// TIA Portal V20 export
ORGANIZATION_BLOCK "Startup"   // OB1040, LAD, Startup
TITLE = "Complete Restart"
AUTHOR : ERsystem_FA2_DH. Kim
// stored: AutoNumber false, IsIECCheckEnabled true, Namespace Unit1.Em4, SetENOAutomatically false
   VAR_INPUT
      LostRetentive : Bool;   // True if retentive data are lost
      LostRTC : Bool;   // True if date and time are lost
   END_VAR
BEGIN

REGION Network 1 (SCL): Build the Absolut Reference Designator
   // Set the Absoult Reference Designator in the Config DB
   IF LEN(IN := "Unit1.Em4.Config".em.referenceDesignator.parent) <> 0 THEN
     "Unit1.Em4.Config".em.referenceDesignator.combined := CONCAT_WSTRING(IN1 := "Unit1.Em4.Config".em.referenceDesignator.parent, IN2 := WSTRING#'.', IN3 := "Unit1.Em4.Config".em.referenceDesignator.relative);
   ELSE
     "Unit1.Em4.Config".em.referenceDesignator.combined := "Unit1.Em4.Config".em.referenceDesignator.relative;
   END_IF;
END_REGION

REGION Network 2 (SCL): Assign axes data
   //Assign axes
   "Unit1.Em4.Config".axis[1] := "BA040AZSCDR5_AnodeMainPnp1AxisX";
   "Unit1.Em4.Config".axis[2] := "BA040AZSCDR6_AnodeMainPnp2AxisX";
   "Unit1.Em4.Config".axis[3] := "BA040AZSCDR11_AnodeMainPnp1AxisY";
   "Unit1.Em4.Config".axis[4] := "BA040AZSCDR12_AnodeMainPnp1AxisZ";
   "Unit1.Em4.Config".axis[5] := "BA040AZSCDR14_AnodeMainPnp2AxisZ";
   "Unit1.Em4.Config".axis[6] := "BA040AZSCDR15_AnodeAlignTableAxisX";
   "Unit1.Em4.Config".axis[7] := "BA040AZSCDR16_AnodeAlignTableAxisY1";
   "Unit1.Em4.Config".axis[8] := "BA040AZSCDR17_AnodeAlignTableAxisY2";

   // Config.cam[1] := _.BA030AZSCDR5_AnodeMainPnp1AxisXCamMain;
   // Config.cam[2] := _.BA030AZSCDR6_AnodeMainPnp2AxisXCamMain;
   // Config.cam[3] := _.BA030AZSCDR12_AnodeMainPnp1AxisZCamMain;
   // Config.cam[4] := _.BA030AZSCDR14_AnodeMainPnp2AxisZCamMain;

   "Unit1.Em4.Config".outputCam[1] := "AnodePnP1XFwd";
   "Unit1.Em4.Config".outputCam[2] := "AnodePnP1XBwd";
   "Unit1.Em4.Config".outputCam[3] := "AnodePnP2XFwd";
   "Unit1.Em4.Config".outputCam[4] := "AnodePnP2XBwd";
   "Unit1.Em4.Config".outputCam[5] := "AnodePnPZ1Down1";
   "Unit1.Em4.Config".outputCam[6] := "AnodePnPZ1Up1";
   "Unit1.Em4.Config".outputCam[7] := "AnodePnPZ2Down1";
   "Unit1.Em4.Config".outputCam[8] := "AnodePnPZ2Up1";
   "Unit1.Em4.Config".outputCam[9] := "AnodePnPZ1Down2";
   "Unit1.Em4.Config".outputCam[10] := "AnodePnPZ1Up2";
   "Unit1.Em4.Config".outputCam[11] := "AnodePnPZ2Down2";
   "Unit1.Em4.Config".outputCam[12] := "AnodePnPZ2Up2";
   "Unit1.Em4.Config".outputCam[13] := "AnodePnPZ1SuctionOn";
   "Unit1.Em4.Config".outputCam[14] := "AnodePnPZ1SuctionOff";
   "Unit1.Em4.Config".outputCam[15] := "AnodePnPZ1ReelCutBlow";
   "Unit1.Em4.Config".outputCam[16] := "AnodePnPZ2SuctionOn";
   "Unit1.Em4.Config".outputCam[17] := "AnodePnPZ2SuctionOff";
   "Unit1.Em4.Config".outputCam[18] := "AnodeAlignSuctionOn";
   "Unit1.Em4.Config".outputCam[19] := "AnodeAlignSuctionOff";

   // Assign configuration data of axis

   // FB Enable
   "Unit1.Em4.HmiInterface".cmAnodeMainPnP1AxisX.commands.enableMasterControl := TRUE;
   "Unit1.Em4.HmiInterface".cmAnodeMainPnP1AxisY.commands.enableMasterControl := TRUE;
   "Unit1.Em4.HmiInterface".cmAnodeMainPnP1AxisZ.commands.enableMasterControl := TRUE;
   "Unit1.Em4.HmiInterface".cmAnodeMainPnP2AxisX.commands.enableMasterControl := TRUE;
   "Unit1.Em4.HmiInterface".cmAnodeMainPnP2AxisZ.commands.enableMasterControl := TRUE;
   "Unit1.Em4.HmiInterface".cmAnodeAlignTableAxisX.commands.enableMasterControl := TRUE;
   "Unit1.Em4.HmiInterface".cmAnodeAlignTableAxisY1.commands.enableMasterControl := TRUE;
   "Unit1.Em4.HmiInterface".cmAnodeAlignTableAxisY2.commands.enableMasterControl := TRUE;

   // Axis 1 BA030AZSCDR5_AnodeMainPnp1AxisX
   "Unit1.Em4.HmiInterface".cmAnodeMainPnP1AxisX.commandConfiguration.jog.velocity := 10.0;
   "Unit1.Em4.HmiInterface".cmAnodeMainPnP1AxisX.commandConfiguration.jog.acceleration := 100.0;
   "Unit1.Em4.HmiInterface".cmAnodeMainPnP1AxisX.commandConfiguration.jog.deceleration := 100.0;
   "Unit1.Em4.HmiInterface".cmAnodeMainPnP1AxisX.commandConfiguration.moveVelocity.velocity := 10.0;
   "Unit1.Em4.HmiInterface".cmAnodeMainPnP1AxisX.commandConfiguration.moveVelocity.acceleration := 100.0;
   "Unit1.Em4.HmiInterface".cmAnodeMainPnP1AxisX.commandConfiguration.moveVelocity.deceleration := 100.0;
   "Unit1.Em4.HmiInterface".cmAnodeMainPnP1AxisX.commandConfiguration.posRelative.velocity := 10.0;
   "Unit1.Em4.HmiInterface".cmAnodeMainPnP1AxisX.commandConfiguration.posRelative.acceleration := 100.0;
   "Unit1.Em4.HmiInterface".cmAnodeMainPnP1AxisX.commandConfiguration.posRelative.deceleration := 100.0;
   "Unit1.Em4.HmiInterface".cmAnodeMainPnP1AxisX.configuration.setPositions[0].name := 'reelCutConveyerPos';
   "Unit1.Em4.HmiInterface".cmAnodeMainPnP1AxisX.configuration.setPositions[1].name := 'alignTablePos';

   // Axis 2 BA030AZSCDR7_AnodeMainPnp2AxisX
   "Unit1.Em4.HmiInterface".cmAnodeMainPnP2AxisX.commandConfiguration.jog.velocity := 10.0;
   "Unit1.Em4.HmiInterface".cmAnodeMainPnP2AxisX.commandConfiguration.jog.acceleration := 100.0;
   "Unit1.Em4.HmiInterface".cmAnodeMainPnP2AxisX.commandConfiguration.jog.deceleration := 100.0;
   "Unit1.Em4.HmiInterface".cmAnodeMainPnP2AxisX.commandConfiguration.moveVelocity.velocity := 10.0;
   "Unit1.Em4.HmiInterface".cmAnodeMainPnP2AxisX.commandConfiguration.moveVelocity.acceleration := 100.0;
   "Unit1.Em4.HmiInterface".cmAnodeMainPnP2AxisX.commandConfiguration.moveVelocity.deceleration := 100.0;
   "Unit1.Em4.HmiInterface".cmAnodeMainPnP2AxisX.commandConfiguration.posRelative.velocity := 10.0;
   "Unit1.Em4.HmiInterface".cmAnodeMainPnP2AxisX.commandConfiguration.posRelative.acceleration := 100.0;
   "Unit1.Em4.HmiInterface".cmAnodeMainPnP2AxisX.commandConfiguration.posRelative.deceleration := 100.0;
   "Unit1.Em4.HmiInterface".cmAnodeMainPnP2AxisX.configuration.setPositions[0].name := 'alignTablePos';
   "Unit1.Em4.HmiInterface".cmAnodeMainPnP2AxisX.configuration.setPositions[1].name := 'stackTablePos';

   // Axis 3 BA030AZSCDR9_AnodeMainPnp1AxisY
   "Unit1.Em4.HmiInterface".cmAnodeMainPnP1AxisY.commandConfiguration.jog.velocity := 10.0;
   "Unit1.Em4.HmiInterface".cmAnodeMainPnP1AxisY.commandConfiguration.jog.acceleration := 100.0;
   "Unit1.Em4.HmiInterface".cmAnodeMainPnP1AxisY.commandConfiguration.jog.deceleration := 100.0;
   "Unit1.Em4.HmiInterface".cmAnodeMainPnP1AxisY.commandConfiguration.moveVelocity.velocity := 10.0;
   "Unit1.Em4.HmiInterface".cmAnodeMainPnP1AxisY.commandConfiguration.moveVelocity.acceleration := 100.0;
   "Unit1.Em4.HmiInterface".cmAnodeMainPnP1AxisY.commandConfiguration.moveVelocity.deceleration := 100.0;
   "Unit1.Em4.HmiInterface".cmAnodeMainPnP1AxisY.commandConfiguration.posRelative.velocity := 10.0;
   "Unit1.Em4.HmiInterface".cmAnodeMainPnP1AxisY.commandConfiguration.posRelative.acceleration := 100.0;
   "Unit1.Em4.HmiInterface".cmAnodeMainPnP1AxisY.commandConfiguration.posRelative.deceleration := 100.0;
   "Unit1.Em4.HmiInterface".cmAnodeMainPnP1AxisY.configuration.setPositions[0].name := 'waitPos';

   // Axis 4 BA030AZSCDR10_AnodeMainPnp1AxisZ
   "Unit1.Em4.HmiInterface".cmAnodeMainPnP1AxisZ.commandConfiguration.jog.velocity := 10.0;
   "Unit1.Em4.HmiInterface".cmAnodeMainPnP1AxisZ.commandConfiguration.jog.acceleration := 100.0;
   "Unit1.Em4.HmiInterface".cmAnodeMainPnP1AxisZ.commandConfiguration.jog.deceleration := 100.0;
   "Unit1.Em4.HmiInterface".cmAnodeMainPnP1AxisZ.commandConfiguration.moveVelocity.velocity := 10.0;
   "Unit1.Em4.HmiInterface".cmAnodeMainPnP1AxisZ.commandConfiguration.moveVelocity.acceleration := 100.0;
   "Unit1.Em4.HmiInterface".cmAnodeMainPnP1AxisZ.commandConfiguration.moveVelocity.deceleration := 100.0;
   "Unit1.Em4.HmiInterface".cmAnodeMainPnP1AxisZ.commandConfiguration.posRelative.velocity := 10.0;
   "Unit1.Em4.HmiInterface".cmAnodeMainPnP1AxisZ.commandConfiguration.posRelative.acceleration := 100.0;
   "Unit1.Em4.HmiInterface".cmAnodeMainPnP1AxisZ.commandConfiguration.posRelative.deceleration := 100.0;
   "Unit1.Em4.HmiInterface".cmAnodeMainPnP1AxisZ.configuration.setPositions[0].name := 'upPos';
   "Unit1.Em4.HmiInterface".cmAnodeMainPnP1AxisZ.configuration.setPositions[1].name := 'reelCutConveyerDownPos';
   "Unit1.Em4.HmiInterface".cmAnodeMainPnP1AxisZ.configuration.setPositions[2].name := 'ailgnTableDownPos';

   // Axis 5 BA030AZSCDR13_AnodeMainPnp2AxisZ
   "Unit1.Em4.HmiInterface".cmAnodeMainPnP2AxisZ.commandConfiguration.jog.velocity := 10.0;
   "Unit1.Em4.HmiInterface".cmAnodeMainPnP2AxisZ.commandConfiguration.jog.acceleration := 100.0;
   "Unit1.Em4.HmiInterface".cmAnodeMainPnP2AxisZ.commandConfiguration.jog.deceleration := 100.0;
   "Unit1.Em4.HmiInterface".cmAnodeMainPnP2AxisZ.commandConfiguration.moveVelocity.velocity := 10.0;
   "Unit1.Em4.HmiInterface".cmAnodeMainPnP2AxisZ.commandConfiguration.moveVelocity.acceleration := 100.0;
   "Unit1.Em4.HmiInterface".cmAnodeMainPnP2AxisZ.commandConfiguration.moveVelocity.deceleration := 100.0;
   "Unit1.Em4.HmiInterface".cmAnodeMainPnP2AxisZ.commandConfiguration.posRelative.velocity := 10.0;
   "Unit1.Em4.HmiInterface".cmAnodeMainPnP2AxisZ.commandConfiguration.posRelative.acceleration := 100.0;
   "Unit1.Em4.HmiInterface".cmAnodeMainPnP2AxisZ.commandConfiguration.posRelative.deceleration := 100.0;
   "Unit1.Em4.HmiInterface".cmAnodeMainPnP2AxisZ.configuration.setPositions[0].name := 'upPos';
   "Unit1.Em4.HmiInterface".cmAnodeMainPnP2AxisZ.configuration.setPositions[1].name := 'ailgnTableDownPos';
   "Unit1.Em4.HmiInterface".cmAnodeMainPnP2AxisZ.configuration.setPositions[2].name := 'stackTableDownPos';

   // Axis 6 BA030AZSCDR15_AnodeAlignTableAxisX
   "Unit1.Em4.HmiInterface".cmAnodeAlignTableAxisX.commandConfiguration.jog.velocity := 10.0;
   "Unit1.Em4.HmiInterface".cmAnodeAlignTableAxisX.commandConfiguration.jog.acceleration := 100.0;
   "Unit1.Em4.HmiInterface".cmAnodeAlignTableAxisX.commandConfiguration.jog.deceleration := 100.0;
   "Unit1.Em4.HmiInterface".cmAnodeAlignTableAxisX.commandConfiguration.moveVelocity.velocity := 10.0;
   "Unit1.Em4.HmiInterface".cmAnodeAlignTableAxisX.commandConfiguration.moveVelocity.acceleration := 100.0;
   "Unit1.Em4.HmiInterface".cmAnodeAlignTableAxisX.commandConfiguration.moveVelocity.deceleration := 100.0;
   "Unit1.Em4.HmiInterface".cmAnodeAlignTableAxisX.commandConfiguration.posRelative.velocity := 10.0;
   "Unit1.Em4.HmiInterface".cmAnodeAlignTableAxisX.commandConfiguration.posRelative.acceleration := 100.0;
   "Unit1.Em4.HmiInterface".cmAnodeAlignTableAxisX.commandConfiguration.posRelative.deceleration := 100.0;
   "Unit1.Em4.HmiInterface".cmAnodeAlignTableAxisX.configuration.setPositions[0].name := 'waitPos';
   "Unit1.Em4.HmiInterface".cmAnodeAlignTableAxisX.configuration.setPositions[1].name := 'adjustPos';

   // Axis 7 BA030AZSCDR16_AnodeAlignTableAxisY1
   "Unit1.Em4.HmiInterface".cmAnodeAlignTableAxisY1.commandConfiguration.jog.velocity := 10.0;
   "Unit1.Em4.HmiInterface".cmAnodeAlignTableAxisY1.commandConfiguration.jog.acceleration := 100.0;
   "Unit1.Em4.HmiInterface".cmAnodeAlignTableAxisY1.commandConfiguration.jog.deceleration := 100.0;
   "Unit1.Em4.HmiInterface".cmAnodeAlignTableAxisY1.commandConfiguration.moveVelocity.velocity := 10.0;
   "Unit1.Em4.HmiInterface".cmAnodeAlignTableAxisY1.commandConfiguration.moveVelocity.acceleration := 100.0;
   "Unit1.Em4.HmiInterface".cmAnodeAlignTableAxisY1.commandConfiguration.moveVelocity.deceleration := 100.0;
   "Unit1.Em4.HmiInterface".cmAnodeAlignTableAxisY1.commandConfiguration.posRelative.velocity := 10.0;
   "Unit1.Em4.HmiInterface".cmAnodeAlignTableAxisY1.commandConfiguration.posRelative.acceleration := 100.0;
   "Unit1.Em4.HmiInterface".cmAnodeAlignTableAxisY1.commandConfiguration.posRelative.deceleration := 100.0;
   "Unit1.Em4.HmiInterface".cmAnodeAlignTableAxisY1.configuration.setPositions[0].name := 'waitPos';
   "Unit1.Em4.HmiInterface".cmAnodeAlignTableAxisY1.configuration.setPositions[1].name := 'adjustPos';

   // Axis 8 BA030AZSCDR17_AnodeAlignTableAxisY2
   "Unit1.Em4.HmiInterface".cmAnodeAlignTableAxisY2.commandConfiguration.jog.velocity := 10.0;
   "Unit1.Em4.HmiInterface".cmAnodeAlignTableAxisY2.commandConfiguration.jog.acceleration := 100.0;
   "Unit1.Em4.HmiInterface".cmAnodeAlignTableAxisY2.commandConfiguration.jog.deceleration := 100.0;
   "Unit1.Em4.HmiInterface".cmAnodeAlignTableAxisY2.commandConfiguration.moveVelocity.velocity := 10.0;
   "Unit1.Em4.HmiInterface".cmAnodeAlignTableAxisY2.commandConfiguration.moveVelocity.acceleration := 100.0;
   "Unit1.Em4.HmiInterface".cmAnodeAlignTableAxisY2.commandConfiguration.moveVelocity.deceleration := 100.0;
   "Unit1.Em4.HmiInterface".cmAnodeAlignTableAxisY2.commandConfiguration.posRelative.velocity := 10.0;
   "Unit1.Em4.HmiInterface".cmAnodeAlignTableAxisY2.commandConfiguration.posRelative.acceleration := 100.0;
   "Unit1.Em4.HmiInterface".cmAnodeAlignTableAxisY2.commandConfiguration.posRelative.deceleration := 100.0;
   "Unit1.Em4.HmiInterface".cmAnodeAlignTableAxisY2.configuration.setPositions[0].name := 'waitPos';
   "Unit1.Em4.HmiInterface".cmAnodeAlignTableAxisY2.configuration.setPositions[1].name := 'adjustPos';
END_REGION

REGION Network 3 (SCL): Assign TwoWayActuator data
   //Assign Configuration data of TwoWayActuator

   //cmAnodeMainPnP1RotaryCwCcw
   "Unit1.Em4.Config".cmAnodeMainPnP1RotaryCwCcw.referenceDesignator := WSTRING#'MainPnP1RotaryCwCcw';
   "Unit1.Em4.Config".cmAnodeMainPnP1RotaryCwCcw.disableFeedbackHomePos := FALSE;
   "Unit1.Em4.Config".cmAnodeMainPnP1RotaryCwCcw.disableFeedbackWorkPos := FALSE;
   "Unit1.Em4.HmiInterface".cmAnodeMainPnP1RotaryCwCcw.configuration.referenceDesignator := WSTRING#'MainPnP1RotaryCwCcw';
   "Unit1.Em4.HmiInterface".cmAnodeMainPnP1RotaryCwCcw.configuration.disableFeedbackHomePos := FALSE;
   "Unit1.Em4.HmiInterface".cmAnodeMainPnP1RotaryCwCcw.configuration.disableFeedbackWorkPos := FALSE;

   //cmAnodeMainPnP1SuctionPlateVacuum
   "Unit1.Em4.Config".cmAnodeMainPnP1SuctionPlateVacuum.referenceDesignator := WSTRING#'MainPnP1Vacuum';
   "Unit1.Em4.Config".cmAnodeMainPnP1SuctionPlateVacuum.disableFeedbackHomePos := FALSE;
   "Unit1.Em4.Config".cmAnodeMainPnP1SuctionPlateVacuum.disableFeedbackWorkPos := FALSE;
   "Unit1.Em4.HmiInterface".cmAnodeMainPnP1SuctionPlateVacuum.configuration.referenceDesignator := WSTRING#'MainPnP1Vacuum';
   "Unit1.Em4.HmiInterface".cmAnodeMainPnP1SuctionPlateVacuum.configuration.disableFeedbackHomePos := FALSE;
   "Unit1.Em4.HmiInterface".cmAnodeMainPnP1SuctionPlateVacuum.configuration.disableFeedbackWorkPos := FALSE;

   //cmAnodeMainPnP2SuctionPlateVacuum
   "Unit1.Em4.Config".cmAnodeMainPnP2SuctionPlateVacuum.referenceDesignator := WSTRING#'MainPnP2Vacuum';
   "Unit1.Em4.Config".cmAnodeMainPnP2SuctionPlateVacuum.disableFeedbackHomePos := FALSE;
   "Unit1.Em4.Config".cmAnodeMainPnP2SuctionPlateVacuum.disableFeedbackWorkPos := FALSE;
   "Unit1.Em4.HmiInterface".cmAnodeMainPnP2SuctionPlateVacuum.configuration.referenceDesignator := WSTRING#'MainPnP2Vacuum';
   "Unit1.Em4.HmiInterface".cmAnodeMainPnP2SuctionPlateVacuum.configuration.disableFeedbackHomePos := FALSE;
   "Unit1.Em4.HmiInterface".cmAnodeMainPnP2SuctionPlateVacuum.configuration.disableFeedbackWorkPos := FALSE;

   //cmAnodeAlignTableSuctionPlateVacuum
   "Unit1.Em4.Config".cmAnodeAlignTableSuctionPlateVacuum.referenceDesignator := WSTRING#'AlignTableVaccum';
   "Unit1.Em4.Config".cmAnodeAlignTableSuctionPlateVacuum.disableFeedbackHomePos := FALSE;
   "Unit1.Em4.Config".cmAnodeAlignTableSuctionPlateVacuum.disableFeedbackWorkPos := FALSE;
   "Unit1.Em4.HmiInterface".cmAnodeAlignTableSuctionPlateVacuum.configuration.referenceDesignator := WSTRING#'AlignTableVaccum';
   "Unit1.Em4.HmiInterface".cmAnodeAlignTableSuctionPlateVacuum.configuration.disableFeedbackHomePos := FALSE;
   "Unit1.Em4.HmiInterface".cmAnodeAlignTableSuctionPlateVacuum.configuration.disableFeedbackWorkPos := FALSE;

   //cmAnodeGlassCleaning
   "Unit1.Em4.Config".cmAnodeGlassCleaning.referenceDesignator := WSTRING#'GlassCleaning';
   "Unit1.Em4.Config".cmAnodeGlassCleaning.disableFeedbackHomePos := TRUE;
   "Unit1.Em4.Config".cmAnodeGlassCleaning.disableFeedbackWorkPos := TRUE;
   "Unit1.Em4.HmiInterface".cmAnodeGlassCleaning.configuration.referenceDesignator := WSTRING#'GlassCleaning';
   "Unit1.Em4.HmiInterface".cmAnodeGlassCleaning.configuration.disableFeedbackHomePos := TRUE;
   "Unit1.Em4.HmiInterface".cmAnodeGlassCleaning.configuration.disableFeedbackWorkPos := TRUE;

   //cmAnodeNgPnpUpDown
   "Unit1.Em4.Config".cmAnodeNgPnpUpDown.referenceDesignator := WSTRING#'NgPnpUpDown';
   "Unit1.Em4.Config".cmAnodeNgPnpUpDown.disableFeedbackHomePos := FALSE;
   "Unit1.Em4.Config".cmAnodeNgPnpUpDown.disableFeedbackWorkPos := FALSE;
   "Unit1.Em4.HmiInterface".cmAnodeNgPnpUpDown.configuration.referenceDesignator := WSTRING#'NgPnpUpDown';
   "Unit1.Em4.HmiInterface".cmAnodeNgPnpUpDown.configuration.disableFeedbackHomePos := FALSE;
   "Unit1.Em4.HmiInterface".cmAnodeNgPnpUpDown.configuration.disableFeedbackWorkPos := FALSE;

   //cmAnodeNgPnp1stFwdBwd
   "Unit1.Em4.Config".cmAnodeNgPnp1stFwdBwd.referenceDesignator := WSTRING#'NgPnp1stFwdBwd';
   "Unit1.Em4.Config".cmAnodeNgPnp1stFwdBwd.disableFeedbackHomePos := FALSE;
   "Unit1.Em4.Config".cmAnodeNgPnp1stFwdBwd.disableFeedbackWorkPos := FALSE;
   "Unit1.Em4.HmiInterface".cmAnodeNgPnp1stFwdBwd.configuration.referenceDesignator := WSTRING#'NgPnp1stFwdBwd';
   "Unit1.Em4.HmiInterface".cmAnodeNgPnp1stFwdBwd.configuration.disableFeedbackHomePos := FALSE;
   "Unit1.Em4.HmiInterface".cmAnodeNgPnp1stFwdBwd.configuration.disableFeedbackWorkPos := FALSE;

   //cmAnodeNgPnp2ndFwdBwd
   "Unit1.Em4.Config".cmAnodeNgPnp2ndFwdBwd.referenceDesignator := WSTRING#'NgPnp2ndFwdBwd';
   "Unit1.Em4.Config".cmAnodeNgPnp2ndFwdBwd.disableFeedbackHomePos := FALSE;
   "Unit1.Em4.Config".cmAnodeNgPnp2ndFwdBwd.disableFeedbackWorkPos := FALSE;
   "Unit1.Em4.HmiInterface".cmAnodeNgPnp2ndFwdBwd.configuration.referenceDesignator := WSTRING#'NgPnp2ndFwdBwd';
   "Unit1.Em4.HmiInterface".cmAnodeNgPnp2ndFwdBwd.configuration.disableFeedbackHomePos := FALSE;
   "Unit1.Em4.HmiInterface".cmAnodeNgPnp2ndFwdBwd.configuration.disableFeedbackWorkPos := FALSE;

   //cmAnodeMaintenanceMovingFixFrontRearFwdBwd
   "Unit1.Em4.Config".cmAnodeMaintenanceMovingFixFrontRearFwdBwd.referenceDesignator := WSTRING#'MaintenanceFix';
   "Unit1.Em4.Config".cmAnodeMaintenanceMovingFixFrontRearFwdBwd.disableFeedbackHomePos := FALSE;
   "Unit1.Em4.Config".cmAnodeMaintenanceMovingFixFrontRearFwdBwd.disableFeedbackWorkPos := FALSE;
   "Unit1.Em4.HmiInterface".cmAnodeMaintenanceMovingFixFrontRearFwdBwd.configuration.referenceDesignator := WSTRING#'MaintenanceFix';
   "Unit1.Em4.HmiInterface".cmAnodeMaintenanceMovingFixFrontRearFwdBwd.configuration.disableFeedbackHomePos := FALSE;
   "Unit1.Em4.HmiInterface".cmAnodeMaintenanceMovingFixFrontRearFwdBwd.configuration.disableFeedbackWorkPos := FALSE;

   //cmAnodeNgBoxLiftUpDown
   "Unit1.Em4.Config".cmAnodeNgBoxLiftUpDown.referenceDesignator := WSTRING#'NgBoxLiftUpDown';
   "Unit1.Em4.Config".cmAnodeNgBoxLiftUpDown.disableFeedbackHomePos := FALSE;
   "Unit1.Em4.Config".cmAnodeNgBoxLiftUpDown.disableFeedbackWorkPos := FALSE;
   "Unit1.Em4.HmiInterface".cmAnodeNgBoxLiftUpDown.configuration.referenceDesignator := WSTRING#'NgBoxLiftUpDown';
   "Unit1.Em4.HmiInterface".cmAnodeNgBoxLiftUpDown.configuration.disableFeedbackHomePos := FALSE;
   "Unit1.Em4.HmiInterface".cmAnodeNgBoxLiftUpDown.configuration.disableFeedbackWorkPos := FALSE;

   //cmAnodeNgBoxLockUpDown
   "Unit1.Em4.Config".cmAnodeNgBoxLockUpDown.referenceDesignator := WSTRING#'NgBoxLockUpDown';
   "Unit1.Em4.Config".cmAnodeNgBoxLockUpDown.disableFeedbackHomePos := FALSE;
   "Unit1.Em4.Config".cmAnodeNgBoxLockUpDown.disableFeedbackWorkPos := FALSE;
   "Unit1.Em4.HmiInterface".cmAnodeNgBoxLockUpDown.configuration.referenceDesignator := WSTRING#'NgBoxLockUpDown';
   "Unit1.Em4.HmiInterface".cmAnodeNgBoxLockUpDown.configuration.disableFeedbackHomePos := FALSE;
   "Unit1.Em4.HmiInterface".cmAnodeNgBoxLockUpDown.configuration.disableFeedbackWorkPos := FALSE;

   //cmAnodeNgPnpVaccum
   "Unit1.Em4.Config".cmAnodeNgPnpVaccum.referenceDesignator := WSTRING#'NgPnpVaccum';
   "Unit1.Em4.Config".cmAnodeNgPnpVaccum.disableFeedbackHomePos := FALSE;
   "Unit1.Em4.Config".cmAnodeNgPnpVaccum.disableFeedbackWorkPos := FALSE;
   "Unit1.Em4.HmiInterface".cmAnodeNgPnpVaccum.configuration.referenceDesignator := WSTRING#'NgPnpVaccum';
   "Unit1.Em4.HmiInterface".cmAnodeNgPnpVaccum.configuration.disableFeedbackHomePos := FALSE;
   "Unit1.Em4.HmiInterface".cmAnodeNgPnpVaccum.configuration.disableFeedbackWorkPos := FALSE;

   //cmAnodeConveyorCoverFwdBwd
   "Unit1.Em4.Config".cmAnodeConveyorCoverFwdBwd.referenceDesignator := WSTRING#'ConveyorCoverFwdBwd';
   "Unit1.Em4.Config".cmAnodeConveyorCoverFwdBwd.disableFeedbackHomePos := FALSE;
   "Unit1.Em4.Config".cmAnodeConveyorCoverFwdBwd.disableFeedbackWorkPos := FALSE;
   "Unit1.Em4.HmiInterface".cmAnodeConveyorCoverFwdBwd.configuration.referenceDesignator := WSTRING#'ConveyorCoverFwdBwd';
   "Unit1.Em4.HmiInterface".cmAnodeConveyorCoverFwdBwd.configuration.disableFeedbackHomePos := FALSE;
   "Unit1.Em4.HmiInterface".cmAnodeConveyorCoverFwdBwd.configuration.disableFeedbackWorkPos := FALSE;

   //cmAnodeConveyorPickUpBlower
   "Unit1.Em4.Config".cmAnodeConveyorPickUpBlower.referenceDesignator := WSTRING#'ConveyorPickUpBlower';
   "Unit1.Em4.Config".cmAnodeConveyorPickUpBlower.disableFeedbackHomePos := TRUE;
   "Unit1.Em4.Config".cmAnodeConveyorPickUpBlower.disableFeedbackWorkPos := TRUE;
   "Unit1.Em4.Config".cmAnodeConveyorPickUpBlower.setOutputHomeContinuously := FALSE;
   "Unit1.Em4.Config".cmAnodeConveyorPickUpBlower.setOutputWorkContinuously := FALSE;
   "Unit1.Em4.Config".cmAnodeConveyorPickUpBlower.monitoringLeavingFeedback := T#100ms;
   "Unit1.Em4.Config".cmAnodeConveyorPickUpBlower.monitoringReachingFeedback := T#100ms;
   "Unit1.Em4.HmiInterface".cmAnodeConveyorPickUpBlower.configuration.referenceDesignator := WSTRING#'ConveyorPickUpBlower';
   "Unit1.Em4.HmiInterface".cmAnodeConveyorPickUpBlower.configuration.disableFeedbackHomePos := TRUE;
   "Unit1.Em4.HmiInterface".cmAnodeConveyorPickUpBlower.configuration.disableFeedbackWorkPos := TRUE;
END_REGION
END_ORGANIZATION_BLOCK
